# EPICS autosave request: iocBoot/iocLinux/built_settings.req
$(P)userCalcEnable
$(P)userCalcOutEnable
$(P)userStringCalcEnable
$(P)userArrayCalcEnable
$(P)userTranEnable
$(P)userAveEnable
$(P)userStringSeqEnable
